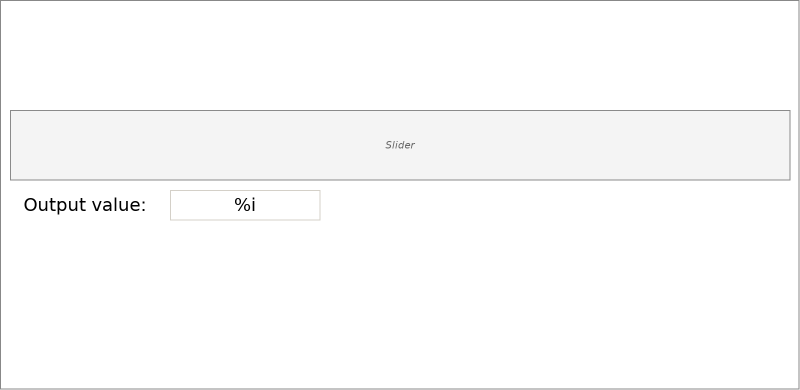
VISUALIZATION VisuAnalogOutControl  // 800x390
VAR_IN_OUT
	pDev : POINTER TO FB_DevAnalogOutput;
END_VAR
    Slider (10,110 780x70), variable: pDev^.fCmdValue, scale 0..100
    Textfield (170,190 150x30), "%i", text variable: pDev^.fCmdValue
        OnMouseClick: write the text variable via VisuDialogs.Numpad
    Label (10,190 150x30), "Output value:"
END_VISUALIZATION

(* stored: Version 1.1.0.1, ProductVersion 3.1.4024.11
   Visu VisuAnalogOutControl: Id {413a08b8-6895-0136-3c12-4d27cfcf25cb} *)
